SYSTEM TL_Task1aDistrA (* System Configuration *)
  (* Standard: 61499-1 *)
  (* Version 0.4, 2009-03-05, JHC, Holobloc Inc., Deleted Application. *)
  (* Version 0.3, 2003-12-05, JHC, Rockwell Automation, Renamed from NEWSYSTEM. *)
  (* Version 0.2, 2002-11-05, JHC, Rockwell Automation, Fixed missing (empty) FBD in Application. *)
  (* Version 0.1, 2002-01-17, JHC, Rockwell Automation, Minor cleanup *)
  (* Version 0.0, 2000-05-27, JHC, Rockwell Automation *)
  PACKAGE fb.rt.myfb;
  IMPORT fb.datatype.*;
  IMPORT fb.rt.*;
  IMPORT fb.rt.events.E_RESTART;
  IMPORT fb.rt.hmi.FRAME_DEVICE;
  IMPORT java.awt.*;
  DEVICE HMI : FRAME_DEVICE(BOUNDS := [0,0,300,300])
    RESOURCE TL1_HMI : VIEW_PANEL(DIA := 5, SIZE := [50,30])
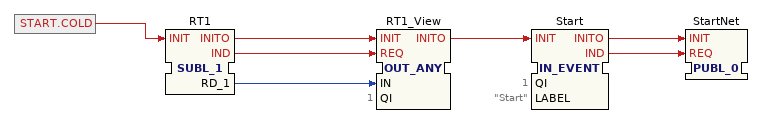
      FBS
        RT1 : SUBL_1;
        RT1_View : OUT_ANY(QI := 1);
        Start : IN_EVENT(QI := 1, LABEL := "Start");
        StartNet : PUBL_0;
      END_FBS
      EVENT_CONNECTIONS
        RT1.INITO TO RT1_View.INIT;
        RT1.IND TO RT1_View.REQ;
        RT1_View.INITO TO Start.INIT;
        Start.INITO TO StartNet.INIT;
        Start.IND TO StartNet.REQ;
        START.COLD TO RT1.INIT;
      END_CONNECTIONS
      DATA_CONNECTIONS
        RT1.RD_1 TO RT1_View.IN;
      END_CONNECTIONS
    END_RESOURCE
    RESOURCE TL2_HMI : VIEW_PANEL(DIA := 5, SIZE := [50,30])
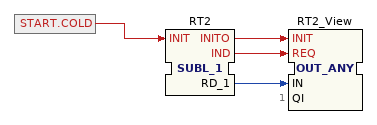
      FBS
        RT2 : SUBL_1;
        RT2_View : OUT_ANY(QI := 1);
      END_FBS
      EVENT_CONNECTIONS
        RT2.INITO TO RT2_View.INIT;
        RT2.IND TO RT2_View.REQ;
        START.COLD TO RT2.INIT;
      END_CONNECTIONS
      DATA_CONNECTIONS
        RT2.RD_1 TO RT2_View.IN;
      END_CONNECTIONS
    END_RESOURCE
  END_DEVICE
  DEVICE VIEW : FRAME_DEVICE(BOUNDS := [300,0,300,300])
    RESOURCE TL1_View : VIEW_PANEL(DIA := 5, SIZE := [50,30])
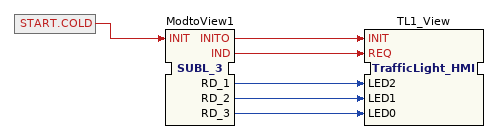
      FBS
        TL1_View : TrafficLight_HMI;
        ModtoView1 : SUBL_3;
      END_FBS
      EVENT_CONNECTIONS
        START.COLD TO ModtoView1.INIT;
        ModtoView1.INITO TO TL1_View.INIT;
        ModtoView1.IND TO TL1_View.REQ;
      END_CONNECTIONS
      DATA_CONNECTIONS
        ModtoView1.RD_1 TO TL1_View.LED2;
        ModtoView1.RD_2 TO TL1_View.LED1;
        ModtoView1.RD_3 TO TL1_View.LED0;
      END_CONNECTIONS
    END_RESOURCE
    RESOURCE TL2_View : VIEW_PANEL(DIA := 5, SIZE := [50,30])
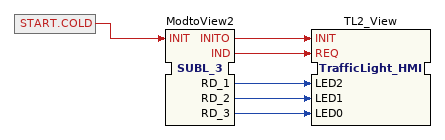
      FBS
        TL2_View : TrafficLight_HMI;
        ModtoView2 : SUBL_3;
      END_FBS
      EVENT_CONNECTIONS
        START.COLD TO ModtoView2.INIT;
        ModtoView2.INITO TO TL2_View.INIT;
        ModtoView2.IND TO TL2_View.REQ;
      END_CONNECTIONS
      DATA_CONNECTIONS
        ModtoView2.RD_1 TO TL2_View.LED2;
        ModtoView2.RD_2 TO TL2_View.LED1;
        ModtoView2.RD_3 TO TL2_View.LED0;
      END_CONNECTIONS
    END_RESOURCE
  END_DEVICE
  DEVICE MODEL : FRAME_DEVICE(BOUNDS := [0,300,300,300])
    RESOURCE TL1_Model : VIEW_PANEL(SIZE := [10,10])
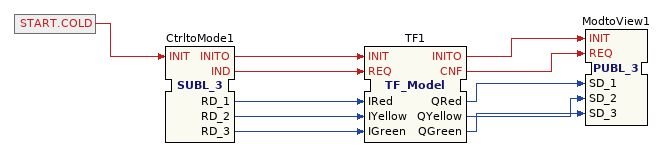
      FBS
        TF1 : TF_Model;
        CtrltoMode1 : SUBL_3;
        ModtoView1 : PUBL_3;
      END_FBS
      EVENT_CONNECTIONS
        START.COLD TO CtrltoMode1.INIT;
        CtrltoMode1.INITO TO TF1.INIT;
        CtrltoMode1.IND TO TF1.REQ;
        TF1.INITO TO ModtoView1.INIT;
        TF1.CNF TO ModtoView1.REQ;
      END_CONNECTIONS
      DATA_CONNECTIONS
        CtrltoMode1.RD_1 TO TF1.IRed;
        CtrltoMode1.RD_2 TO TF1.IYellow;
        CtrltoMode1.RD_3 TO TF1.IGreen;
        TF1.QRed TO ModtoView1.SD_1;
        TF1.QYellow TO ModtoView1.SD_2;
        TF1.QGreen TO ModtoView1.SD_3;
      END_CONNECTIONS
    END_RESOURCE
    RESOURCE TL2_Model : VIEW_PANEL(SIZE := [10,10])
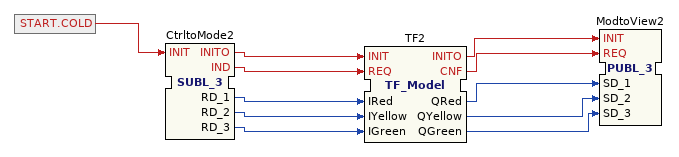
      FBS
        TF2 : TF_Model;
        ModtoView2 : PUBL_3;
        CtrltoMode2 : SUBL_3;
      END_FBS
      EVENT_CONNECTIONS
        TF2.INITO TO ModtoView2.INIT;
        TF2.CNF TO ModtoView2.REQ;
        CtrltoMode2.INITO TO TF2.INIT;
        CtrltoMode2.IND TO TF2.REQ;
        START.COLD TO CtrltoMode2.INIT;
      END_CONNECTIONS
      DATA_CONNECTIONS
        TF2.QRed TO ModtoView2.SD_1;
        TF2.QYellow TO ModtoView2.SD_2;
        TF2.QGreen TO ModtoView2.SD_3;
        CtrltoMode2.RD_1 TO TF2.IRed;
        CtrltoMode2.RD_2 TO TF2.IYellow;
        CtrltoMode2.RD_3 TO TF2.IGreen;
      END_CONNECTIONS
    END_RESOURCE
  END_DEVICE
  DEVICE CONTROLLER : FRAME_DEVICE(BOUNDS := [300,300,300,300])
    RESOURCE Control1 : VIEW_PANEL(SIZE := [10,10])
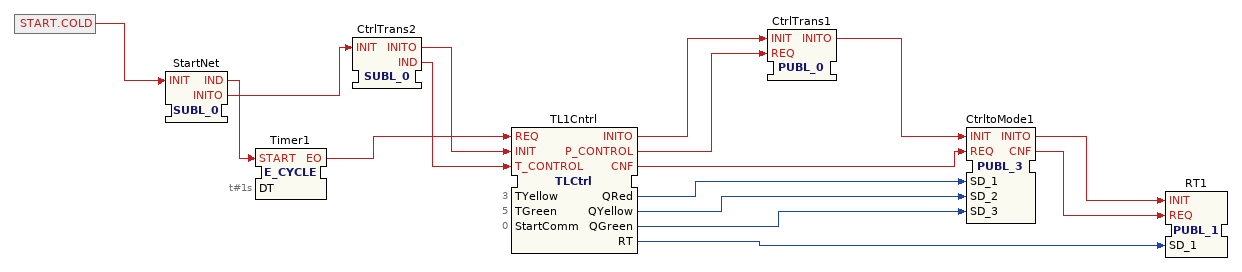
      FBS
        TL1Cntrl : TLCtrl(TYellow := 3, TGreen := 5, StartComm := 0);
        Timer1 : E_CYCLE(DT := t#1s);
        CtrltoMode1 : PUBL_3;
        RT1 : PUBL_1;
        StartNet : SUBL_0;
        CtrlTrans1 : PUBL_0;
        CtrlTrans2 : SUBL_0;
      END_FBS
      EVENT_CONNECTIONS
        CtrltoMode1.INITO TO RT1.INIT;
        CtrltoMode1.CNF TO RT1.REQ;
        START.COLD TO StartNet.INIT;
        StartNet.IND TO Timer1.START;
        Timer1.EO TO TL1Cntrl.REQ;
        TL1Cntrl.INITO TO CtrlTrans1.INIT;
        CtrlTrans1.INITO TO CtrltoMode1.INIT;
        StartNet.INITO TO CtrlTrans2.INIT;
        CtrlTrans2.INITO TO TL1Cntrl.INIT;
        CtrlTrans2.IND TO TL1Cntrl.T_CONTROL;
        TL1Cntrl.P_CONTROL TO CtrlTrans1.REQ;
        TL1Cntrl.CNF TO CtrltoMode1.REQ;
      END_CONNECTIONS
      DATA_CONNECTIONS
        TL1Cntrl.QRed TO CtrltoMode1.SD_1;
        TL1Cntrl.QYellow TO CtrltoMode1.SD_2;
        TL1Cntrl.QGreen TO CtrltoMode1.SD_3;
        TL1Cntrl.RT TO RT1.SD_1;
      END_CONNECTIONS
    END_RESOURCE
    RESOURCE Control2 : VIEW_PANEL(SIZE := [10,10])
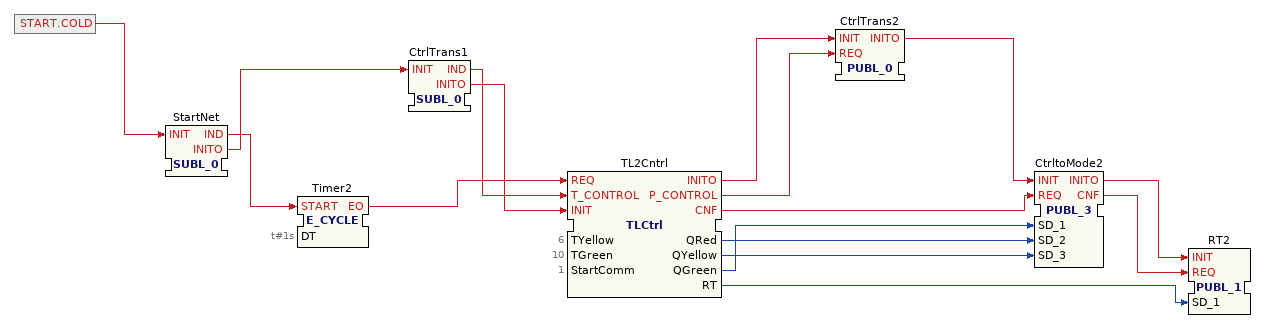
      FBS
        Timer2 : E_CYCLE(DT := t#1s);
        TL2Cntrl : TLCtrl(TYellow := 6, TGreen := 10, StartComm := 1);
        CtrltoMode2 : PUBL_3;
        RT2 : PUBL_1;
        StartNet : SUBL_0;
        CtrlTrans2 : PUBL_0;
        CtrlTrans1 : SUBL_0;
      END_FBS
      EVENT_CONNECTIONS
        CtrltoMode2.INITO TO RT2.INIT;
        CtrltoMode2.CNF TO RT2.REQ;
        START.COLD TO StartNet.INIT;
        StartNet.IND TO Timer2.START;
        Timer2.EO TO TL2Cntrl.REQ;
        TL2Cntrl.INITO TO CtrlTrans2.INIT;
        CtrlTrans2.INITO TO CtrltoMode2.INIT;
        StartNet.INITO TO CtrlTrans1.INIT;
        CtrlTrans1.IND TO TL2Cntrl.T_CONTROL;
        TL2Cntrl.P_CONTROL TO CtrlTrans2.REQ;
        TL2Cntrl.CNF TO CtrltoMode2.REQ;
        CtrlTrans1.INITO TO TL2Cntrl.INIT;
      END_CONNECTIONS
      DATA_CONNECTIONS
        TL2Cntrl.QRed TO CtrltoMode2.SD_1;
        TL2Cntrl.QYellow TO CtrltoMode2.SD_2;
        TL2Cntrl.QGreen TO CtrltoMode2.SD_3;
        TL2Cntrl.RT TO RT2.SD_1;
      END_CONNECTIONS
    END_RESOURCE
  END_DEVICE
END_SYSTEM
